{attribute 'no_check'}
//Generates a pulse signal 
FUNCTION_BLOCK Pulse
VAR_INPUT
	IN														: BOOL; //Start pulse generator
	PT_ON													: TIME; //Time pulse on	
	PT_OFF													: TIME; //Time pulse off 
END_VAR             										
VAR_OUTPUT          										
	Q														: BOOL; 
	RT														: BOOL; 
	FT														: BOOL;
END_VAR             										
VAR                 	
	TON_PULSE												: TON;
END_VAR

	(* Pulse generator																*)
	(********************************************************************************)

(* Reset flag *)
RT := FT													:= FALSE;
(* logic *)
IF 	Q AND(TON_PULSE.Q OR NOT IN)
THEN
	TON_PULSE(IN:=FALSE  , PT:= PT_OFF);
	FT 														:= Q;
	Q 														:= FALSE;
ELSIF NOT Q AND TON_PULSE.Q
	OR_ELSE In AND NOT TON_PULSE.IN 
THEN
	RT 														:= NOT Q;
	TON_PULSE(IN:= FALSE , PT:= PT_ON) ;
	Q 														:= TRUE;
END_IF

//Run timer
TON_PULSE(IN:=IN);

(***********************************************************************************************************************)

END_FUNCTION_BLOCK

(* stored: Version 1.1.0.1, ProductVersion 3.1.4024.3
   POU Pulse: Id {2a50aa56-d732-42b9-9a11-566ccd23cd33}, SpecialFunc None *)
